TYPE ST_EL1809 :
STRUCT
	//--------------------------------------------------------------------------------------------------------
	sTerminalName                                           :   STRING(200):= 'EL1809 | 16-Channel Digital Input';
    //============================================================================================================================	
	// TERMINAL - EL1809 16-Channel Digital Input Terminal (Term 8)	
	iStartButoon                			AT %I*			: 	BOOL;	// EL1809 channel 1
	iStopButton                   			AT %I*			: 	BOOL;	// EL1809 channel 2
	iUP_OK        							AT %I*	 		: 	BOOL;	// EL1809 channel 3
	iUS_OK		   							AT %I*	 		: 	BOOL;	// EL1809 channel 4
	iPartPresentNest1         				AT %I*	 		: 	BOOL;	// EL1809 channel 5 		     			
	iPartPresentNest2 						AT %I*			: 	BOOL;	// EL1809 channel 6
	iEL1809_Ch7               				AT %I*          :   BOOL;   // EL1809 channel 7 
    iEL1809_Ch8          					AT %I*          :   BOOL;   // EL1809 channel 8
    iEL1809_Ch9           					AT %I*          :   BOOL;   // EL1809 channel 9
	iProcessCylinderExtended              	AT %I*          :   BOOL;   // EL1809 channel 10
	iRejectSensor              				AT %I*          :   BOOL;   // EL1809 channel 11
	iEL1809_Ch12			              	AT %I*          :   BOOL;   // EL1809 channel 12	   
	iEL1809_Ch13         		   			AT %I*	 		: 	BOOL;	// EL1809 channel 13   
	iEL1809_Ch14       						AT %I*	 		: 	BOOL;	// EL1809 channel 14 
	iPuckSensorUp	(*Renan Added 06/07*)	AT %I*			: 	BOOL;	// EL1809 channel 15  
	iPuckSensorDown	(*Renan Added 06/07*)	AT %I*	 		: 	BOOL;	// EL1809 channel 16  	
	
	stTerminalInfo											: 	ST_Terminal_Info;

END_STRUCT
END_TYPE

(* stored: Version 1.1.0.1, ProductVersion 3.1.4026.17
   DUT ST_EL1809: Id {75a73e5d-4ca3-4f42-b76f-6978af3e18bb} *)
